{attribute 'OPC.UA.DA.StructuredType' := '1'}
TYPE ST_ActiveStorageSystemState :
STRUCT
	bLoading : BOOL;
END_STRUCT
END_TYPE

(* stored: Version 1.1.0.1, ProductVersion 3.1.4024.10
   DUT ST_ActiveStorageSystemState: Id {b0ef14c6-cc4c-45d0-a615-b8de1b3df083} *)
